SUBAPPLICATION mapping (* Subapplication Type *)
  (* Standard: 61499-2 *)
  (* Version 1.0, 2023-02-19, franz *)
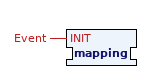
  EVENT_INPUT
    INIT;
  END_EVENT
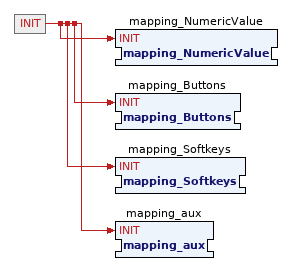
  SUBAPPS
    mapping_NumericValue : mapping_NumericValue;
    mapping_Softkeys : mapping_Softkeys;
    mapping_Buttons : mapping_Buttons;
    mapping_aux : mapping_aux;
  END_SUBAPPS
  EVENT_CONNECTIONS
    INIT TO mapping_NumericValue.INIT;
    INIT TO mapping_Softkeys.INIT;
    INIT TO mapping_Buttons.INIT;
    INIT TO mapping_aux.INIT;
  END_CONNECTIONS
END_SUBAPPLICATION
